(* IEC 61131-3 sources: ConveyorControl-with-PLC/4E_Gruppe1_Graf_Projekt1/Class/_DriveMng_MDD100, 1 file *)

(* ---- _DriveMng_MDD100.st ---- *)
(*!
<Class
	Name               = "_DriveMng_MDD100"
	Revision           = "1.54"
	RealtimeTask       = "false"
	CyclicTask         = "true"
	DefCyclictime      = "10 ms"
	BackgroundTask     = "false"
	Sigmatek           = "true"
	OSInterface        = "false"
	HighPriority       = "false"
	Automatic          = "false"
	UpdateMode         = "Prescan"
	IconPath           = ".\Class\_DriveMngBase\Drive.ico"
	SharedCommandTable = "true"
	Objectsize         = "(586,120)"
	Comment            = "manages the whole varancommunication between&#13;&#10;the Drive and the application">
	<Channels>
		<Server Name="CRC_ErrorCounter" Visualized="true" Initialize="false" WriteProtected="true" Retentive="false" Comment="counts the CRC errors of all axis"/>
		<Server Name="FwDate" Class="VirtualBaseInit" Visualized="false" Initialize="true" WriteProtected="true" Retentive="false" Comment="use this channel to access the string functions"/>
		<Server Name="FWVersion" Class="VirtualBaseInit" Visualized="false" Initialize="true" WriteProtected="true" Retentive="false" Comment="use this channel to access the string functions"/>
		<Server Name="Input1" Visualized="true" Initialize="false" WriteProtected="true" Retentive="false" Comment="State of digital input 1 of drive&#13;&#10;&#13;&#10;-1..input information not available&#13;&#10; 0..input is low&#13;&#10; 1..input is high"/>
		<Server Name="Input2" Visualized="true" Initialize="false" WriteProtected="true" Retentive="false" Comment="State of digital input 2 of drive&#13;&#10;&#13;&#10;-1..input information not available&#13;&#10; 0..input is low&#13;&#10; 1..input is high"/>
		<Server Name="Input3" Visualized="true" Initialize="false" WriteProtected="true" Retentive="false" Comment="State of digital input 3 of drive&#13;&#10;&#13;&#10;-1..input information not available&#13;&#10; 0..input is low&#13;&#10; 1..input is high"/>
		<Server Name="Input4" Visualized="true" Initialize="false" WriteProtected="true" Retentive="false" Comment="State of digital input 4 of drive&#13;&#10;&#13;&#10;-1..input information not available&#13;&#10; 0..input is low&#13;&#10; 1..input is high"/>
		<Server Name="Input5" Visualized="true" Initialize="false" WriteProtected="true" Retentive="false" Comment="State of digital input 5 of drive&#13;&#10;&#13;&#10;-1..input information not available&#13;&#10; 0..input is low&#13;&#10; 1..input is high"/>
		<Server Name="Input6" Visualized="true" Initialize="false" WriteProtected="true" Retentive="false" Comment="State of digital input 6 of drive&#13;&#10;&#13;&#10;-1..input information not available&#13;&#10; 0..input is low&#13;&#10; 1..input is high"/>
		<Server Name="Input7" Visualized="true" Initialize="false" WriteProtected="true" Retentive="false" Comment="State of digital input 7 of drive&#13;&#10;&#13;&#10;-1..input information not available&#13;&#10; 0..input is low&#13;&#10; 1..input is high"/>
		<Server Name="Input8" Visualized="true" Initialize="false" WriteProtected="true" Retentive="false" Comment="State of digital input 8 of drive&#13;&#10;&#13;&#10;-1..input information not available&#13;&#10; 0..input is low&#13;&#10; 1..input is high"/>
		<Server Name="ValidateSerNo" Visualized="true" Initialize="false" WriteProtected="false" Retentive="false" Comment="if the validation of the serial number is activated (SerNoValidation = 1)&#13;&#10;the serial number of the actual module can be validated by writing to this server&#13;&#10;&#13;&#10;this server shows also the state of validation:&#13;&#10;-2..validation not acivated&#13;&#10;-1..no module validated on this position&#13;&#10; 0..module is not the validated one&#13;&#10; 1..module is the validated one"/>
		<Server Name="VaranOut_1" Class="Hub_Base" Visualized="true" Initialize="false" WriteProtected="true" Retentive="false" Comment="VaranOut"/>
		<Client Name="FetchDigitalInputs" Required="false" Internal="false" Comment="Client is set as init value.&#13;&#10;a value &lt;&gt; 0 means the digital inputs of the drive are fetched synchronously and displayed on the Servers Input1 to Input8&#13;&#10;If the function is active an additional VARAN object is used"/>
		<Client Name="FWDateString" Required="true" Internal="true"/>
		<Client Name="FWNumSTring" Required="true" Internal="true"/>
		<Client Name="Required" Required="true" Internal="false" Comment="0=module is not required, 1=module is required "/>
		<Client Name="SerNoValidation" Required="false" Internal="false" Comment="0..serial number of varan client does not matter&#13;&#10;1..serial number of varan client has to be validated, to use the module&#13;&#10;&#13;&#10;validation is done via write(1) to the ValidateSerNo Server"/>
		<Client Name="Transparent" Required="false" Internal="false" DefValue="0" Comment="If this Client is set to 1 the module is not used for building the VARAN-Tree"/>
		<Client Name="UserAction" Required="false" Internal="false" Comment="optional, connect to server to get Varan states (connect,disconnect,interrupt)"/>
		<Client Name="VaranDriveBase" Required="true" Internal="true"/>
		<Client Name="VaranIn" Required="true" Internal="false" Comment="Connect with a Varan Communication Class"/>
		<Client Name="VaranTimeMultiplier" Required="false" Internal="false" Comment="multiplier of varan time set as init value."/>
	</Channels>
	<RevDoku>
		<Owner Company="Sigmatek" Author="WalRob"/>
		<Dokumentation Revision="1.54" Date="25.08.2015" Author="EisMic" Company="Sigmatek" Description="DataObjects are now installed in UpdateCy and are added to DOList in UpdateRt if the OS supports the new interface method. Version 16#1003 or higher of the pMultiVaran-Interface is needed to use this feature."/>
		<Dokumentation Revision="1.53" Date="18.06.2015" Author="PieSte" Company="Sigmatek" Description="Add newinst command to call methode DisableDevice() and EnableDevice() to avoid retrys when hw disconnected.&#13;&#10;Corrected function Varan_HwDisconnect() to set dataobjects off."/>
		<Dokumentation Revision="1.52" Date="26.05.2015" Author="RamAnd" Company="Sigmatek" Description="Added possibility to get enabled Axis which is needed to set absolute position of axis."/>
		<Dokumentation Revision="1.51" Date="16.04.2015" Author="PieSte&#13;&#10;LanSte&#13;&#10;PieSte" Company="Sigmatek" Description="Added support for visualisation in graphical hardware editor.&#13;&#10;Added support for calculating resources for graphical hardware editor.&#13;&#10;Add new parameter to read drive scope faster. It is used for SDD1X00 drives."/>
		<Dokumentation Revision="1.50" Date="24.03.2015" Author="EisMic" Company="Sigmatek" Description="Check pointer p_NodeInfo for validity in method GetRetryTimeout due to access exception error if method Varan_HWDisconnect is called and no hardware was available."/>
		<Dokumentation Revision="1.49" Date="06.03.2015" Author="PieSte" Company="Sigmatek" Description="Changed commands for businterface to be compatible with new drive hardware.&#13;&#10;Changed visual state of FwNumString and FwDateString object for lse displaying."/>
		<Dokumentation Revision="1.48" Date="27.01.2015" Author="EisMic" Company="Sigmatek" Description="Implemented commando for lasal 2 to get serial number of drive."/>
		<Dokumentation Revision="1.47" Date="13.08.2014" Author="LanSte" Company="Sigmatek" Description="Corrected reading Firmwareversion with newinst cmd: CMD_GET_HARDWARE_DIAGNOSE "/>
		<Dokumentation Revision="1.46" Date="30.07.2014" Author="RamAnd" Company="Sigmatek" Description="Loop to check for retries could have caused a crash, if the drive wasn&apos;t initialized so far."/>
		<Dokumentation Revision="1.45" Date="25.07.2014" Author="LanSte&#13;&#10;PieSte" Company="Sigmatek" Description="Added Support for reading hardware diagnose and hardwaretree entry.&#13;&#10;Corrected internal call of GetParameterState in baseclass _DriveMngBase."/>
		<Dokumentation Revision="1.44" Date="04.07.2014" Author="PieSte" Company="Sigmatek" Description="Saved client FetchDigitalInputs to TempFetchDigitalInputs in baseclass to avoid an access exception if it is changed during run."/>
		<Dokumentation Revision="1.43" Date="07.05.2014" Author="EisMic" Company="Sigmatek" Description="Added missing servers in lhd file and corrected the type of servers."/>
		<Dokumentation Revision="1.42" Date="07.05.2014" Author="LanSte" Company="Sigmatek" Description="Improved Transparent property description in HW-Tree and activated greying out of the object in the HW-Tree.&#13;&#10;Minimized the interface request via CILGET by useing private pointers to reduce time in init."/>
		<Dokumentation Revision="1.41" Date="06.03.2014" Author="RamAnd" Company="Sigmatek" Description="Changed offset of SyncOut 1 (62,5µs) to be synchron with the SyncOut 0 to prevent inconsistent data in the drive firmware."/>
		<Dokumentation Revision="1.40" Date="12.02.2014" Author="ZoePat&#13;&#10;ZoePat" Company="Sigmatek" Description="Added new NewInst comando for Lasal2 to get the list of axis.&#13;&#10;ExtendedAxis for Axis2 of SDD210 and SDD215 din&apos;t work."/>
		<Dokumentation Revision="1.30" Date="20.01.2014" Author="RamAnd&#13;&#10;&#13;&#10;PieSte" Company="Sigmatek" Description="Success of GetSyncParameter and SetSyncParameter couldn&apos;t be ensured because the return value wasn&apos;t initialized if the method succeeds.&#13;&#10;Add TaskDelay 15ms in _VaranDriveBase Varan_HwConnect to initialize the Hardware."/>
		<Dokumentation Revision="1.20" Date="05.12.2013" Author="LanSte" Company="Sigmatek" Description="Added payload support"/>
		<Dokumentation Revision="1.10" Date="05.11.2012" Author="RamAnd" Company="Sigmatek" Description="Content of corresponding LASAL Hardware Description file (.lhd) which is necessary for the hardware editor has been updated"/>
		<Dokumentation Revision="1.8" Date="02.11.2011" Author="SvePau" Company="Sigmatek" Description="Changed comment of the Client &quot;FetchDigitalInputs&quot; and added possibility to set it via HW-Editor"/>
		<Dokumentation Revision="1.7" Date="05.08.2011" Author="PibPet" Company="Sigmatek" Description="Input Server changed Visulized to TRUE SA:19236"/>
		<Dokumentation Revision="1.6" Date="28.06.2011" Author="BleErn" Company="Sigmatek" Description="Content of corresponding LASAL Hardware Description file (.lhd) which is necessary for the hardware editor has been updated"/>
		<Dokumentation Revision="1.5" Date="15.06.2011" Author="Ramand" Company="Sigmatek" Description="Client Transparent has to be not required, as it is a new feature."/>
		<Dokumentation Revision="1.4" Date="31.05.2011" Author="RamAnd" Company="Sigmatek" Description="Added possibility to read out the digital inputs of the drive synchronously."/>
		<Dokumentation Revision="1.3" Date="18.05.2011" Author="RamAnd" Company="Sigmatek" Description="After the Online-Server changed to 1, it was possible that the synchron values (like actual position) took 1 more realtime cycle to be shown by the class."/>
		<Dokumentation Revision="1.2" Date="20.04.2011" Author="SvePau" Company="Sigmatek" Description="Connected server ValidateSerNo from baseclass to derivation"/>
		<Dokumentation Revision="1.1" Date="13.04.2011" Author="BleErn" Company="Sigmatek" Description="Added Client Transparent that allows to disable a VARAN-HW-Class"/>
		<Dokumentation Revision="1.0" Date="09.02.2011" Author="WalRob" Company="Sigmatek" Description="Initial version"/>
	</RevDoku>
	<Network Name="_DriveMng_MDD100">
		<!-- List of Components in this network -->
		<Components>
			<Object
				Name       = "_base"
				Class      = "_DriveMngBase"
				Position   = "(1816,120)"
				Visualized = "false">
				<Channels>
					<Server Name="AxisAvailable"/>
					<Server Name="CmdState"/>
					<Server Name="DeviceAddress"/>
					<Server Name="DeviceID"/>
					<Server Name="DriveType"/>
					<Server Name="HWVersion"/>
					<Server Name="Online"/>
					<Server Name="Release"/>
					<Server Name="RetryCounter"/>
					<Server Name="SerialNo"/>
					<Server Name="VendorID"/>
					<Client Name="cOnline"/>
					<Client Name="coStdLib"/>
					<Client Name="FwDatetr"/>
					<Client Name="FwNumStr"/>
					<Client Name="To_TaskObjectControl"/>
					<Client Name="ToBusIF"/>
					<Client Name="toVaran"/>
				</Channels>
			</Object>
			<Object
				Name       = "FWDateString"
				Class      = "String"
				Position   = "(1170,450)"
				Visualized = "true">
				<Channels>
					<Server Name="Data"/>
					<Client Name="SingleRealloc" Value="1"/>
				</Channels>
			</Object>
			<Object
				Name       = "FWNumSTring"
				Class      = "String"
				Position   = "(1170,300)"
				Visualized = "true">
				<Channels>
					<Server Name="Data"/>
					<Client Name="SingleRealloc" Value="1"/>
				</Channels>
			</Object>
			<Object
				Name       = "VaranDriveBase"
				Class      = "_VaranDriveBase"
				Position   = "(450,120)"
				Visualized = "false">
				<Channels>
					<Server Name="CRC_ErrorCounter"/>
					<Server Name="DeviceAddress"/>
					<Server Name="DeviceID"/>
					<Server Name="Input1"/>
					<Server Name="Input2"/>
					<Server Name="Input3"/>
					<Server Name="Input4"/>
					<Server Name="Input5"/>
					<Server Name="Input6"/>
					<Server Name="Input7"/>
					<Server Name="Input8"/>
					<Server Name="Online"/>
					<Server Name="Release"/>
					<Server Name="RetryCounter"/>
					<Server Name="SerialNo"/>
					<Server Name="State"/>
					<Server Name="Synchron"/>
					<Server Name="ValidateSerNo"/>
					<Server Name="VaranOut_1"/>
					<Server Name="VendorID"/>
					<Client Name="FetchDigitalInputs" Value="0"/>
					<Client Name="Required" Value="1"/>
					<Client Name="SerNoValidation"/>
					<Client Name="Transparent" Value="0"/>
					<Client Name="UserAction"/>
					<Client Name="VaranIn"/>
					<Client Name="VaranTimeMultiplier"/>
				</Channels>
			</Object>
		</Components>
		<Comments>
		</Comments>
		<!-- List of Connections in this network -->
		<Connections>
			<Connection Source="this.CmdState" Destination="_base.CmdState" Vertices="(2478,210),(2306,210),"/>
			<Connection Source="VaranDriveBase.VaranIn" Destination="this.VaranIn" Vertices="(450,210),(120,210),(120,810),(38,810),"/>
			<Connection Source="VaranDriveBase.Required" Destination="this.Required" Vertices="(450,270),(180,270),(180,870),(38,870),"/>
			<Connection Source="this.VaranDriveBase" Destination="VaranDriveBase.State"/>
			<Connection Source="VaranDriveBase.VaranTimeMultiplier" Destination="this.VaranTimeMultiplier" Vertices="(450,510),(300,510),(300,1110),(38,1110),"/>
			<Connection Source="VaranDriveBase.UserAction" Destination="this.UserAction" Vertices="(450,330),(210,330),(210,930),(38,930),"/>
			<Connection Source="_base.toVaran" Destination="VaranDriveBase.State" Vertices="(1816,210),(1050,210),"/>
			<Connection Source="_base.cOnline" Destination="VaranDriveBase.Online" Vertices="(1816,270),(1050,270),"/>
			<Connection Source="this.Online" Destination="_base.Online" Vertices="(2478,270),(2306,270),"/>
			<Connection Source="this.Release" Destination="_base.Release" Vertices="(2478,330),(2306,330),"/>
			<Connection Source="this.DriveType" Destination="_base.DriveType" Vertices="(2478,630),(2306,630),"/>
			<Connection Source="this.DeviceAddress" Destination="_base.DeviceAddress" Vertices="(2478,390),(2306,390),"/>
			<Connection Source="this.VendorID" Destination="_base.VendorID" Vertices="(2478,450),(2306,450),"/>
			<Connection Source="this.DeviceID" Destination="_base.DeviceID" Vertices="(2478,510),(2306,510),"/>
			<Connection Source="this.RetryCounter" Destination="_base.RetryCounter" Vertices="(2478,570),(2306,570),"/>
			<Connection Source="this.SerialNo" Destination="_base.SerialNo" Vertices="(2478,690),(2340,690),(2306,750),"/>
			<Connection Source="_base.FwDatetr" Destination="FWDateString.Data" Vertices="(1816,390),(1710,390),(1710,450),(1710,540),(1486,540),"/>
			<Connection Source="this.HWVersion" Destination="_base.HWVersion" Vertices="(2478,750),(2340,750),(2306,810),"/>
			<Connection Source="this.CRC_ErrorCounter" Destination="VaranDriveBase.CRC_ErrorCounter" Vertices="(2478,990),(1170,990),(1170,750),(1050,750),"/>
			<Connection Source="this.VaranOut_1" Destination="VaranDriveBase.VaranOut_1" Vertices="(2478,1530),(1110,1530),(1110,1350),(1050,1350),"/>
			<Connection Source="this.FWNumSTring" Destination="FWNumSTring.Data"/>
			<Connection Source="this.FWDateString" Destination="FWDateString.Data"/>
			<Connection Source="this.FwDate" Destination="FWDateString.Data" Vertices="(2478,870),(2340,870),(2310,900),(1530,900),(1530,540),(1486,540),"/>
			<Connection Source="_base.FwNumStr" Destination="FWNumSTring.Data" Vertices="(1816,330),(1560,330),(1560,390),(1486,390),"/>
			<Connection Source="this.FWVersion" Destination="FWNumSTring.Data" Vertices="(2478,810),(2340,810),(2310,870),(1560,870),(1560,390),(1486,390),"/>
			<Connection Source="VaranDriveBase.SerNoValidation" Destination="this.SerNoValidation" Vertices="(450,390),(240,390),(240,990),(38,990),"/>
			<Connection Source="VaranDriveBase.Transparent" Destination="this.Transparent" Vertices="(450,450),(270,450),(270,1050),(38,1050),"/>
			<Connection Source="this.ValidateSerNo" Destination="VaranDriveBase.ValidateSerNo" Vertices="(2478,930),(1200,930),(1200,690),(1050,690),"/>
			<Connection Source="VaranDriveBase.FetchDigitalInputs" Destination="this.FetchDigitalInputs" Vertices="(450,570),(330,570),(330,1170),(38,1170),"/>
			<Connection Source="this.Input1" Destination="VaranDriveBase.Input1" Vertices="(2478,1050),(1140,1050),(1140,870),(1050,870),"/>
			<Connection Source="this.Input2" Destination="VaranDriveBase.Input2" Vertices="(2478,1110),(1140,1110),(1140,930),(1050,930),"/>
			<Connection Source="this.Input3" Destination="VaranDriveBase.Input3" Vertices="(2478,1170),(1140,1170),(1140,990),(1050,990),"/>
			<Connection Source="this.Input4" Destination="VaranDriveBase.Input4" Vertices="(2478,1230),(1140,1230),(1140,1050),(1050,1050),"/>
			<Connection Source="this.Input5" Destination="VaranDriveBase.Input5" Vertices="(2478,1290),(1140,1290),(1140,1110),(1050,1110),"/>
			<Connection Source="this.Input6" Destination="VaranDriveBase.Input6" Vertices="(2478,1350),(1140,1350),(1140,1170),(1050,1170),"/>
			<Connection Source="this.Input7" Destination="VaranDriveBase.Input7" Vertices="(2478,1410),(1140,1410),(1140,1230),(1050,1230),"/>
			<Connection Source="this.Input8" Destination="VaranDriveBase.Input8" Vertices="(2478,1470),(1140,1470),(1140,1290),(1050,1290),"/>
		</Connections>
		<!-- Headerfiles -->
		<Options>
		</Options>
	</Network>
</Class>
*)
#pragma using _DriveMngBase

_DriveMng_MDD100 : CLASS
: _DriveMngBase
  //Servers:
	FWVersion 	: SvrChCmd_UDINT;
	FwDate 	: SvrChCmd_UDINT;
	ValidateSerNo 	: SvrCh_DINT;
	CRC_ErrorCounter 	: SvrCh_DINT;
	Input1 	: SvrCh_DINT;
	Input2 	: SvrCh_DINT;
	Input3 	: SvrCh_DINT;
	Input4 	: SvrCh_DINT;
	Input5 	: SvrCh_DINT;
	Input6 	: SvrCh_DINT;
	Input7 	: SvrCh_DINT;
	Input8 	: SvrCh_DINT;
	VaranOut_1 	: SvrChCmd_DINT;
  //Clients:
	VaranIn 	: CltChCmd_Hub_Base;
	Required 	: CltCh_DINT;
	UserAction 	: CltCh_DINT;
	SerNoValidation 	: CltCh_DINT;
	Transparent 	: CltCh_DINT;
	VaranTimeMultiplier 	: CltCh_UDINT;
	FWDateString 	: CltChCmd_String;
	FWNumSTring 	: CltChCmd_String;
	VaranDriveBase 	: CltChCmd__VaranDriveBase;
	FetchDigitalInputs 	: CltCh_DINT;
  //Variables:
  //Functions:

	FUNCTION VIRTUAL GetBusDeviceID
		VAR_OUTPUT
			output 	: UDINT;
		END_VAR;

	FUNCTION VIRTUAL GetDrvDeviceID
		VAR_OUTPUT
			output 	: UDINT;
		END_VAR;

	FUNCTION VIRTUAL GLOBAL CRC_ErrorCounter::Read
		VAR_OUTPUT
			output (EAX) 	: DINT;
		END_VAR;

	FUNCTION VIRTUAL GLOBAL Input1::Read
		VAR_OUTPUT
			output (EAX) 	: DINT;
		END_VAR;

	FUNCTION VIRTUAL GLOBAL Input2::Read
		VAR_OUTPUT
			output (EAX) 	: DINT;
		END_VAR;

	FUNCTION VIRTUAL GLOBAL Input3::Read
		VAR_OUTPUT
			output (EAX) 	: DINT;
		END_VAR;

	FUNCTION VIRTUAL GLOBAL Input4::Read
		VAR_OUTPUT
			output (EAX) 	: DINT;
		END_VAR;

	FUNCTION VIRTUAL GLOBAL Input5::Read
		VAR_OUTPUT
			output (EAX) 	: DINT;
		END_VAR;

	FUNCTION VIRTUAL GLOBAL Input6::Read
		VAR_OUTPUT
			output (EAX) 	: DINT;
		END_VAR;

	FUNCTION VIRTUAL GLOBAL Input7::Read
		VAR_OUTPUT
			output (EAX) 	: DINT;
		END_VAR;

	FUNCTION VIRTUAL GLOBAL Input8::Read
		VAR_OUTPUT
			output (EAX) 	: DINT;
		END_VAR;

	FUNCTION VIRTUAL GLOBAL VaranOut_1::Read
		VAR_OUTPUT
			output (EAX) 	: DINT;
		END_VAR;
  //Tables:
	FUNCTION @STD
		VAR_OUTPUT
			ret_code	: CONFSTATES;
		END_VAR;
	FUNCTION GLOBAL TAB @CT_;
END_CLASS;

#pragma using _VaranDriveBase
#pragma using String
#pragma usingLtd Hub_Base

FUNCTION VIRTUAL GLOBAL _DriveMng_MDD100::CRC_ErrorCounter::Read
	VAR_OUTPUT
		output (EAX) 	: DINT;
	END_VAR

	CRC_ErrorCounter := VaranDriveBase.CRC_ErrorCounter.Read();
	output := CRC_ErrorCounter;

END_FUNCTION

FUNCTION VIRTUAL GLOBAL _DriveMng_MDD100::VaranOut_1::Read
	VAR_OUTPUT
		output (EAX) 	: DINT;
	END_VAR

	VaranOut_1 := VaranDriveBase.VaranOut_1.Read();
	output := VaranOut_1;

END_FUNCTION

FUNCTION VIRTUAL GLOBAL _DriveMng_MDD100::Input1::Read
	VAR_OUTPUT
		output (EAX) 	: DINT;
	END_VAR

	Input1 := VaranDriveBase.Input1.Read();
	output := Input1;

END_FUNCTION

FUNCTION VIRTUAL GLOBAL _DriveMng_MDD100::Input2::Read
	VAR_OUTPUT
		output (EAX) 	: DINT;
	END_VAR

	Input2 := VaranDriveBase.Input2.Read();
	output := Input2;

END_FUNCTION

FUNCTION VIRTUAL GLOBAL _DriveMng_MDD100::Input3::Read
	VAR_OUTPUT
		output (EAX) 	: DINT;
	END_VAR

	Input3 := VaranDriveBase.Input3.Read();
	output := Input3;

END_FUNCTION

FUNCTION VIRTUAL GLOBAL _DriveMng_MDD100::Input4::Read
	VAR_OUTPUT
		output (EAX) 	: DINT;
	END_VAR

	Input4 := VaranDriveBase.Input4.Read();
	output := Input4;

END_FUNCTION

FUNCTION VIRTUAL GLOBAL _DriveMng_MDD100::Input5::Read
	VAR_OUTPUT
		output (EAX) 	: DINT;
	END_VAR

	Input5 := VaranDriveBase.Input5.Read();
	output := Input5;

END_FUNCTION

FUNCTION VIRTUAL GLOBAL _DriveMng_MDD100::Input6::Read
	VAR_OUTPUT
		output (EAX) 	: DINT;
	END_VAR

	Input6 := VaranDriveBase.Input6.Read();
	output := Input6;

END_FUNCTION

FUNCTION VIRTUAL GLOBAL _DriveMng_MDD100::Input7::Read
	VAR_OUTPUT
		output (EAX) 	: DINT;
	END_VAR

	Input7 := VaranDriveBase.Input7.Read();
	output := Input7;

END_FUNCTION

FUNCTION VIRTUAL GLOBAL _DriveMng_MDD100::Input8::Read
	VAR_OUTPUT
		output (EAX) 	: DINT;
	END_VAR

	Input8 := VaranDriveBase.Input8.Read();
	output := Input8;

END_FUNCTION

FUNCTION VIRTUAL _DriveMng_MDD100::GetBusDeviceID
	VAR_OUTPUT
		output 	: UDINT;
	END_VAR

  output := DRIVEMNG_BUSDEVICEID_MDD;

END_FUNCTION

FUNCTION VIRTUAL _DriveMng_MDD100::GetDrvDeviceID
	VAR_OUTPUT
		output 	: UDINT;
	END_VAR

  output := DRIVEMNG_DRVDEVICEID_MDD121;

END_FUNCTION
